FUNCTION Convert_ULINT_TO_UINT : Hresult
VAR_INPUT
	in : ULINT;
	out : REFERENCE TO UINT;
END_VAR
VAR
	converted : UINT;
END_VAR
VAR CONSTANT
	INCOMPATIBLE : HRESULT := 16#9811070E;
END_VAR

converted := ULINT_TO_UINT(in);

IF (UINT_TO_ULINT(converted) <> in) THEN
	Convert_ULINT_TO_UINT := INCOMPATIBLE;
	RETURN;
END_IF

out := converted;

END_FUNCTION

(* stored: Version 1.1.0.1, ProductVersion 3.1.4024.12
   POU Convert_ULINT_TO_UINT: Id {bc9db924-86c5-4c59-b876-5c16719f3bad}, SpecialFunc None *)
